TYPE CommandBlockBase :
STRUCT	
	AXIS_ID: WORD;
	COMMAND_TYPE:eCommandTypes;
	SPEED:LWORD; // in 0.001mm
	ACC_TIME:LWORD; // in ms
	DEC_TIME:LWORD; // in ms
	TORQUE_LIMIT:LWORD; // in 0.01 percentage
END_STRUCT
END_TYPE

(* stored: Version 1.1.0.1, ProductVersion 3.1.4022.10
   DUT CommandBlockBase: Id {44762155-a4ee-4688-ad57-0991b5877603} *)
